// TwinCAT 3 PLC project Untitled
// ProgramVersion: 3.1.4023.0
// libraries:
//   Tc2_Standard, * (Beckhoff Automation GmbH)
//   Tc2_System, * (Beckhoff Automation GmbH)
//   Tc3_IoLink, * (Beckhoff Automation GmbH)
//   Tc3_Module, * (Beckhoff Automation GmbH)
// project tree:
//   / PlcTask.TcTTO
//   POUs/ MAIN.TcPOU

CONFIGURATION Untitled
    RESOURCE PLC ON TwinCAT3
        TASK PlcTask(INTERVAL := T#10ms, PRIORITY := 20);
        PROGRAM MAIN WITH PlcTask : MAIN;
    END_RESOURCE
END_CONFIGURATION

// ---- POUs/MAIN.TcPOU
PROGRAM MAIN
VAR
	
	nSwitchCtrl			:	BOOL	:=	TRUE;
	nRotateUpper		:	WORD	:=	16#8000;
	nRotateLower		:	WORD	:=	16#01;
	
	
	bEL6224_Ch1		AT%I*	:	BOOL;
	
	bEL2008_value	AT%Q*	:	BYTE;
	
END_VAR

END_PROGRAM
